{attribute 'qualified_only'}
{attribute 'strict'}
TYPE E_AXIS_MotionType : (
	NONE,
	MCHOME,
	MCVELOCITY,
	MCABSOLUT,
	MCRELATIVE
	//E_AXIS_MCMODULO,
	//E_AXIS_MCHALT,
	//E_AXIS_MCSTOP
);
END_TYPE

(* stored: Version 1.1.0.1
   DUT E_AXIS_MotionType: Id {d89aeb0a-7a1f-4ec1-b9bc-dc442b907187} *)
